FUNCTION fRateLimit : LREAL
VAR_INPUT
END_VAR
VAR
END_VAR

END_FUNCTION

(* stored: Version 1.1.0.1
   POU fRateLimit: Id {ee22e1bc-9072-4895-a5c2-7f8ebd098940}, SpecialFunc None *)
